FUNCTION_BLOCK ForcibleInt_Test
VAR
END_VAR

ForceOff();
ForceOn();
ForcibleAcceptsValue();
ForciblePassesUnforcedValue();

METHOD ForceOff
VAR
	Expected	 : INT;
	Actual		 : INT;
	Forcible : ForcibleInt('');
END_VAR
IF TestSuite.Test(__POUNAME()).ExecuteTest() THEN
	Expected := 0;
	Forcible.SetForceState(E_ForceState.ForceOff);
	Forcible.Input := 12;
	Actual	:= Forcible.Output;
	TestSuite.Test(__POUNAME()).AssertEqual(Expected, Actual);
END_IF
END_METHOD

METHOD ForceOn
VAR
	Expected	 : INT;
	Actual		 : INT;
	Forcible : ForcibleInt('');
END_VAR
IF TestSuite.Test(__POUNAME()).ExecuteTest() THEN
	Expected := 16;
	Forcible.ForceValue := 16;
	Forcible.SetForceState(E_ForceState.ForceOn);
	Forcible.Input := 23;
	Actual			   := Forcible.Output;
	TestSuite.Test(__POUNAME()).AssertEqual(Expected, Actual);
END_IF
END_METHOD

METHOD ForcibleAcceptsValue
VAR
	Expected	 : INT;
	Actual		 : INT;
	Forcible : ForcibleInt('');
END_VAR
IF TestSuite.Test(__POUNAME()).ExecuteTest() THEN
	Expected := 17;
	Forcible.ForceValue := Expected;
	Actual			   := Forcible.ForceValue;
	TestSuite.Test(__POUNAME()).AssertEqual(Expected, Actual);
END_IF
END_METHOD

METHOD ForciblePassesUnforcedValue
VAR
	Expected	 : INT;
	Actual		 : INT;
	Forcible : ForcibleInt('');
END_VAR
IF TestSuite.Test(__POUNAME()).ExecuteTest() THEN
	Expected := 16;
	Forcible.SetForceState(E_ForceState.Unforced);
	Forcible.Input := 16;
	Actual			   := Forcible.Output;
	TestSuite.Test(__POUNAME()).AssertEqual(Expected, Actual);
END_IF
END_METHOD

END_FUNCTION_BLOCK

(* stored: Version 1.1.0.1, ProductVersion 3.1.4026.18
   POU ForcibleInt_Test: Id {2f9cf0f1-d030-45bf-b782-62522d677f5a}, SpecialFunc None
   Method ForceOff: Id {4d4970d2-14e3-4347-b9c3-45b8f984675e}
   Method ForceOn: Id {739f519d-3921-43cd-832e-bfa4947cb96e}
   Method ForcibleAcceptsValue: Id {1f48dbd0-403c-4cdd-af0c-a2434cd9cab7}
   Method ForciblePassesUnforcedValue: Id {c33e2b19-d07b-4d3f-a34a-afe5b49e1799} *)
